// LS Electric XG5000 project: 최종 plc 프레임_변경안1
// PLC LSPLC
// module base 0 slot 0: 입출력 모듈:XBC-DR32H (DC 24V 입력, 릴레이 출력 32점)

PROGRAM NewProgram (task: 스캔 프로그램)

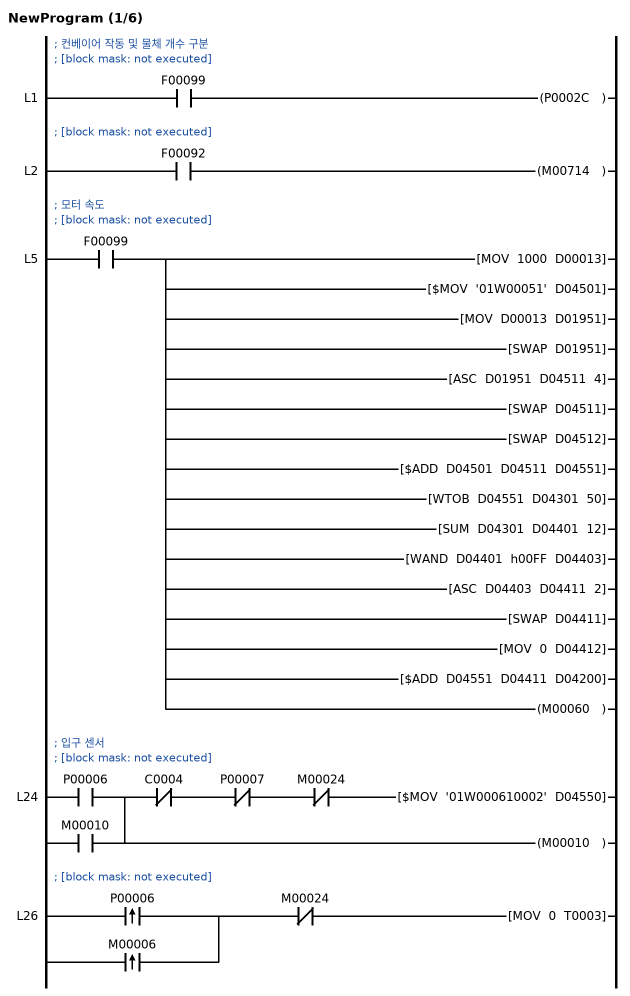
// 컨베이어 작동 및 물체 개수 구분
; L1 (block mask: not executed)
LOAD      F00099
OUT       P0002C
; L2 (block mask: not executed)
LOAD      F00092
OUT       M00714
// 모터 속도
; L5 (block mask: not executed)
LOAD      F00099
MOV       1000 D00013
$MOV      '01W00051' D04501
MOV       D00013 D01951
SWAP      D01951
ASC       D01951 D04511 4
SWAP      D04511
SWAP      D04512
$ADD      D04501 D04511 D04551
WTOB      D04551 D04301 50
SUM       D04301 D04401 12
WAND      D04401 h00FF D04403
ASC       D04403 D04411 2
SWAP      D04411
MOV       0 D04412
$ADD      D04551 D04411 D04200
OUT       M00060
// 입구 센서
; L24 (block mask: not executed)
LOAD      P00006
OR        M00010
MPUSH
AND NOT   C0004
AND NOT   P00007
AND NOT   M00024
$MOV      '01W000610002' D04550
MPOP
OUT       M00010
; L26 (block mask: not executed)
LOADP     P00006
ORP       M00006
AND NOT   M00024
MOV       0 T0003

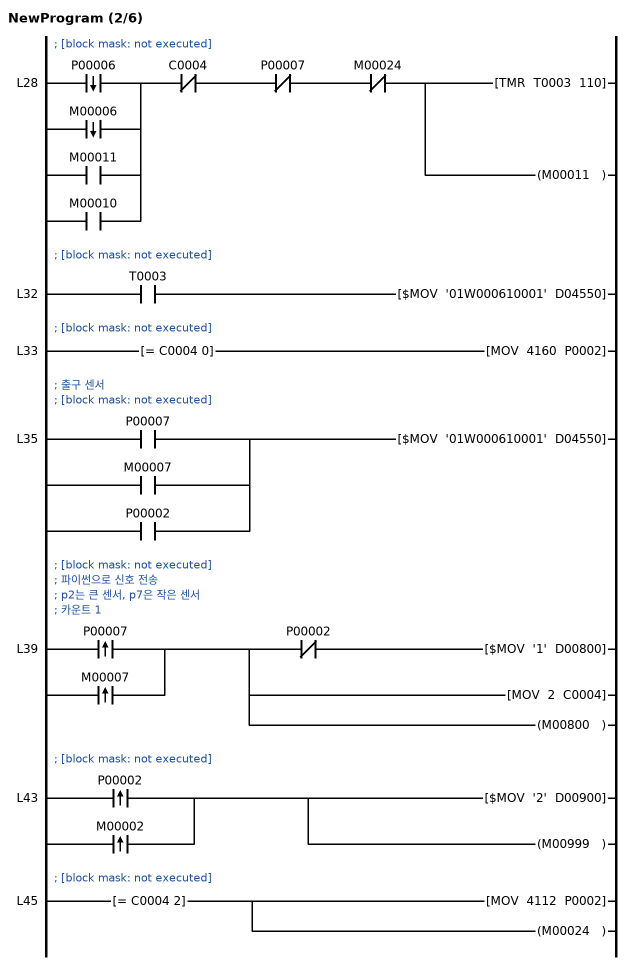
; L28 (block mask: not executed)
LOADN     P00006
ORN       M00006
OR        M00011
OR        M00010
AND NOT   C0004
AND NOT   P00007
AND NOT   M00024
TMR       T0003 110
OUT       M00011
; L32 (block mask: not executed)
LOAD      T0003
$MOV      '01W000610001' D04550
; L33 (block mask: not executed)
LOAD=     C0004 0
MOV       4160 P0002
// 출구 센서
; L35 (block mask: not executed)
LOAD      P00007
OR        M00007
OR        P00002
$MOV      '01W000610001' D04550
; L39 (block mask: not executed)
LOADP     P00007
ORP       M00007
MPUSH
AND NOT   P00002
$MOV      '1' D00800
MPOP
MOV       2 C0004
OUT       M00800
// output comment: 파이썬으로 신호 전송 p2는 큰 센서, p7은 작은 센서
// output comment: 카운트 1
; L43 (block mask: not executed)
LOADP     P00002
ORP       M00002
$MOV      '2' D00900
OUT       M00999
; L45 (block mask: not executed)
LOAD=     C0004 2
MOV       4112 P0002
OUT       M00024

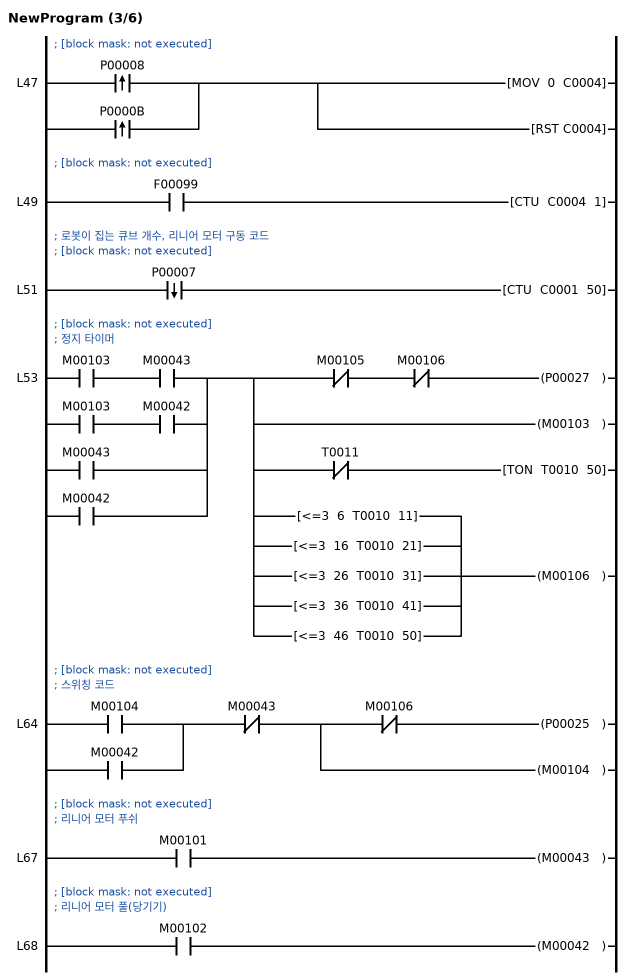
; L47 (block mask: not executed)
LOADP     P00008
ORP       P0000B
MOV       0 C0004
RST       C0004
; L49 (block mask: not executed)
LOAD      F00099
CTU       C0004 1
// 로봇이 집는 큐브 개수, 리니어 모터 구동 코드
; L51 (block mask: not executed)
LOADN     P00007
CTU       C0001 50
; L53 (block mask: not executed)
LOAD      M00103
AND       M00043
LOAD      M00103
AND       M00042
OR LOAD
OR        M00043
OR        M00042
MPUSH
AND NOT   M00105
AND NOT   M00106
OUT       P00027
MLOAD
OUT       M00103
AND NOT   T0011
TON       T0010 50
MPOP
LOAD<=3   6 T0010 11
OR<=3     16 T0010 21
OR<=3     26 T0010 31
OR<=3     36 T0010 41
OR<=3     46 T0010 50
AND LOAD
OUT       M00106
// output comment: 정지 타이머
; L64 (block mask: not executed)
LOAD      M00104
OR        M00042
AND NOT   M00043
MPUSH
AND NOT   M00106
OUT       P00025
MPOP
OUT       M00104
// output comment: 스위칭 코드
; L67 (block mask: not executed)
LOAD      M00101
OUT       M00043
// output comment: 리니어 모터 푸쉬
; L68 (block mask: not executed)
LOAD      M00102
OUT       M00042
// output comment: 리니어 모터 풀(당기기)

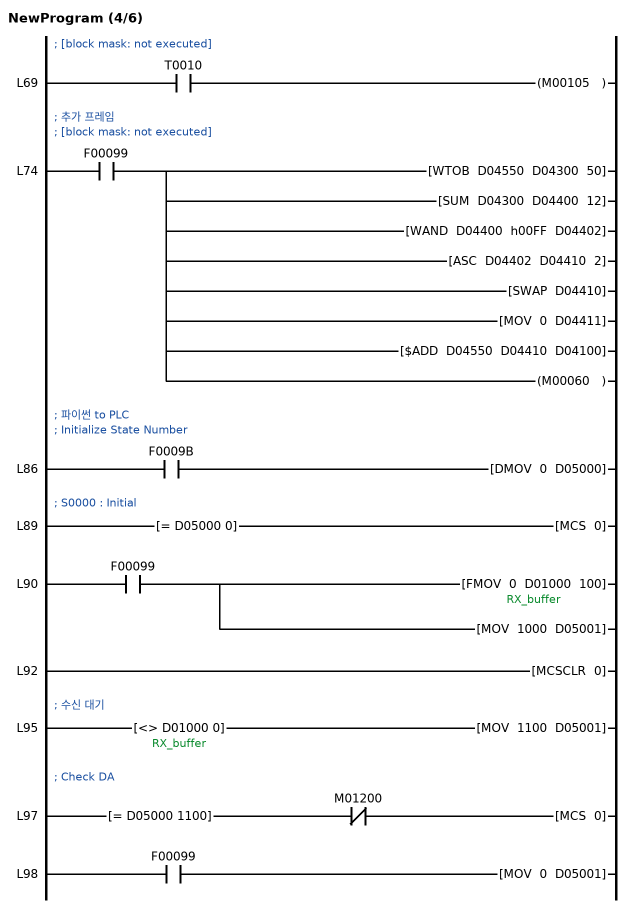
; L69 (block mask: not executed)
LOAD      T0010
OUT       M00105
// 추가 프레임
; L74 (block mask: not executed)
LOAD      F00099
WTOB      D04550 D04300 50
SUM       D04300 D04400 12
WAND      D04400 h00FF D04402
ASC       D04402 D04410 2
SWAP      D04410
MOV       0 D04411
$ADD      D04550 D04410 D04100
OUT       M00060
// 파이썬 to PLC
// Initialize State Number
; L86
LOAD      F0009B
DMOV      0 D05000
// S0000 : Initial
; L89
LOAD=     D05000 0
MCS       0
; L90
LOAD      F00099
FMOV      0 D01000 100	// RX_buffer
MOV       1000 D05001
; L92
MCSCLR    0
// 수신 대기
; L95
LOAD<>    D01000 0	// RX_buffer
MOV       1100 D05001
// Check DA
; L97
LOAD=     D05000 1100
AND NOT   M01200
MCS       0
; L98
LOAD      F00099
MOV       0 D05001

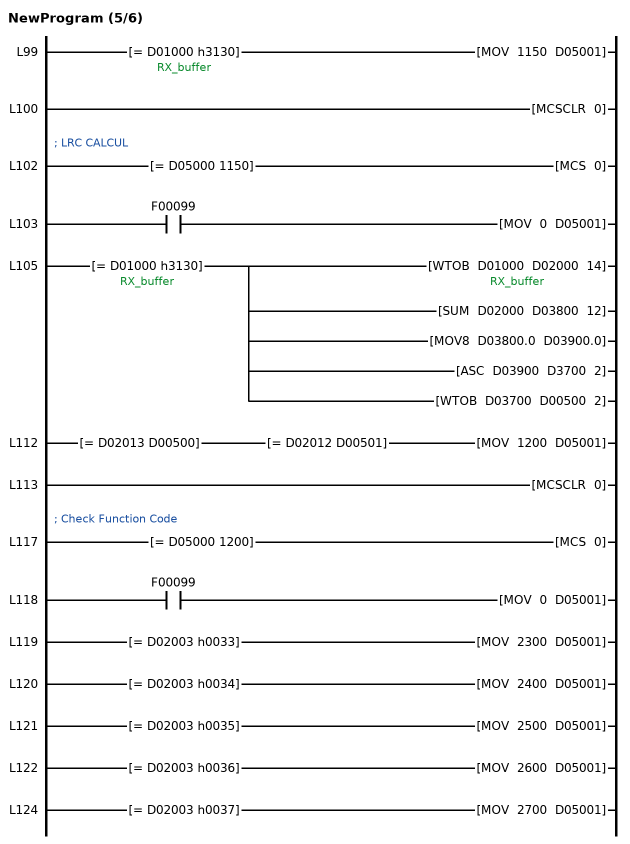
; L99
LOAD=     D01000 h3130	// RX_buffer
MOV       1150 D05001
; L100
MCSCLR    0
// LRC CALCUL
; L102
LOAD=     D05000 1150
MCS       0
; L103
LOAD      F00099
MOV       0 D05001
; L105
LOAD=     D01000 h3130	// RX_buffer
WTOB      D01000 D02000 14	// RX_buffer
SUM       D02000 D03800 12
MOV8      D03800.0 D03900.0
ASC       D03900 D3700 2
WTOB      D03700 D00500 2
; L112
LOAD=     D02013 D00500
AND=      D02012 D00501
MOV       1200 D05001
; L113
MCSCLR    0
// Check Function Code
; L117
LOAD=     D05000 1200
MCS       0
; L118
LOAD      F00099
MOV       0 D05001
; L119
LOAD=     D02003 h0033
MOV       2300 D05001
; L120
LOAD=     D02003 h0034
MOV       2400 D05001
; L121
LOAD=     D02003 h0035
MOV       2500 D05001
; L122
LOAD=     D02003 h0036
MOV       2600 D05001
; L124
LOAD=     D02003 h0037
MOV       2700 D05001

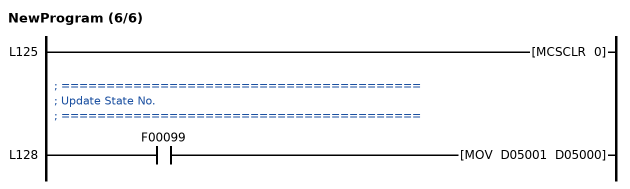
; L125
MCSCLR    0
// ========================================
// Update State No.
// ========================================
; L128
LOAD      F00099
MOV       D05001 D05000

VARIABLES AND COMMENTS (devices not used above)
D00999	WORD	RX